(* PLC project preparation, Dassault Systèmes ControlBuild 2024x *)
(* stored: creationDateTime 2023-10-03T11:13:41-01:00 *)

FUNCTION_BLOCK bottling_line.preparation
  VAR_INPUT
    preparationRequest : BOOL := false;
    productionWaiting : BOOL := false;
  END_VAR
  VAR_INPUT
    highLevel1 : BOOL := false;
    highLevel2 : BOOL := false;
    highLevel3 : BOOL := false;
  END_VAR
  VAR_OUTPUT
    preparationValve1 : BOOL := false;
    preparationValve2 : BOOL := false;
    preparationValve3 : BOOL := false;
    preparationValve4 : BOOL := false;
    preparationPump1 : BOOL := false;
    preparationPump2 : BOOL := false;
    preparationAgit : BOOL := false;
  END_VAR
  VAR_OUTPUT
    preparationEnd : BOOL := false;
  END_VAR

INITIAL_STEP 10:
  COMPUTE_FUNCTION_BLOCKS(S);
END_STEP
TRANSITION FROM 10 TO 11
  := preparationRequest;
END_TRANSITION
STEP 11:
  11_INLINE1(N);
END_STEP
ACTION 11_INLINE1:
  IF NOT highLevel1 THEN
  	preparationValve1;
  END_IF;
  IF NOT highLevel2 THEN
  	preparationValve2;
  END_IF;
END_ACTION
TRANSITION FROM 11 TO 12
  := highLevel1 AND highLevel2;
END_TRANSITION
STEP 12:
  12_INLINE2(N);
END_STEP
ACTION 12_INLINE2:
  preparationAgit;
  preparationPump1;
  preparationPump2;
  preparationValve3;
  preparationValve4;
END_ACTION
TRANSITION FROM 12 TO 13
  := highLevel3;
END_TRANSITION
STEP 13:
  13_INLINE3(N);
END_STEP
ACTION 13_INLINE3:
  preparationEnd;
END_ACTION
TRANSITION FROM 13 TO 10
  := productionWaiting;
END_TRANSITION
ACTION COMPUTE_FUNCTION_BLOCKS:  (* blocks drawn on the SFC sheet *)
  G1:
END_ACTION
END_FUNCTION_BLOCK
